FUNCTION_BLOCK Feeder IMPLEMENTS MachineModule
VAR
	(*General Movement Trigger*)
	bEnable			: BOOL;
	bDisable        : BOOL;
	bError          : BOOL;
	bOverride       : BOOL;
	bSimulation     : BOOL;
	bStart          : BOOL;
	bStop           : BOOL;
	
	(*Sensor Specific Trigger*)
	bBottomHit 		: I_Sensor;
	bTopHit			: I_Sensor;
	(*Internal Variable*)
	nMovement 		: INT;
	nmovetest		: INT;
	(*Fedder*)
	bFeederPlateInPos	: BOOL;

END_VAR

(*Business Logic here*)

IF 	bEnable 
	AND NOT (bError)
	AND nMovement<1500 THEN
	
	nMovement := nMovement+1;
	bStop:=FALSE; (*Could use this thing in another module*)
	
END_IF

IF nMovement=1500 THEN
	bStop:=TRUE;
END_IF

METHOD Disable : BOOL 
VAR_INPUT
END_VAR
bEnable:=FALSE;
END_METHOD

METHOD Enable : BOOL
VAR_INPUT
END_VAR
bEnable:=TRUE;
bDisable:=FALSE;
END_METHOD

METHOD Error : BOOL
VAR_INPUT
END_VAR
bEnable:=FALSE;
END_METHOD

METHOD FB_init : BOOL
VAR_INPUT
	bInitRetains : BOOL; // if TRUE, the retain variables are initialized (warm start / cold start)
	bInCopyCode : BOOL;  // if TRUE, the instance afterwards gets moved into the copy code (online change)
	bBottomHit 		: I_Sensor;
	bTopHit			: I_Sensor;
END_VAR
THIS^.bBottomHit	:= bBottomHit;
THIS^.bTopHit		:= bTopHit;
END_METHOD

METHOD Override : BOOL
VAR_INPUT
END_VAR
END_METHOD

METHOD Reset : BOOL
VAR_INPUT
END_VAR
END_METHOD

METHOD Start : BOOL
VAR_INPUT
END_VAR
END_METHOD

METHOD PUBLIC StateMachine
VAR_INPUT

END_VAR
IF bEnable THEN
	nmovetest:=nmovetest+1;	
	ELSE
		
	nmovetest:=0;
END_IF
END_METHOD

METHOD Stop : BOOL
VAR_INPUT
END_VAR
END_METHOD

END_FUNCTION_BLOCK

(* stored: Version 1.1.0.1, ProductVersion 3.1.4024.12
   POU Feeder: Id {7c4ba1ca-5c7a-4b43-bce2-192dcc10d3e9}, SpecialFunc None
   Method Disable: Id {67148c7b-6ee3-4791-a511-6a80a34ec26c}
   Method Enable: Id {903e6d0b-3746-4369-aebc-bbcba2c3a8d5}
   Method Error: Id {be472e56-0c8b-4050-bec9-f54152999515}
   Method FB_init: Id {02bddd52-7631-4084-83f2-ccba1d5ef21d}
   Method Override: Id {f6a40ca7-f285-41af-ae0b-7138c692a8d3}
   Method Reset: Id {46056118-b452-4d98-8e71-bae590cde4a6}
   Method Start: Id {1f67bb41-f3df-4402-b491-9f139d9e706a}
   Method StateMachine: Id {41ceeb2c-3832-4fa5-b551-06150a392abb}
   Method Stop: Id {f67300df-0080-45fe-b0fb-7c05483d98a3} *)
